{attribute 'qualified_only'}
VAR_GLOBAL
	// Digital Outputs
	bGreenLight 			AT %Q* : BOOL;
	bRedLight 				AT %Q* : BOOL;
	
	// Analog Outputs
	nValveOutput 			AT %Q* : INT; 
END_VAR

(* stored: Version 1.1.0.1, ProductVersion 3.1.4024.13
   GVL G_Output: Id {9f09a37e-4151-41e9-b303-85d293f6f5b3} *)
